DATA_BLOCK "ST10_FB_S7connect_IDB"
{ S7_Optimized_Access := 'TRUE' }
VERSION : 0.1
NON_RETAIN
// ATTRIBUTES
// AUTO_NUMBER = False
// BLOCK_NUMBER = 900
// END_ATTRIBUTES
"ST10_FB_S7connect"

BEGIN

END_DATA_BLOCK

